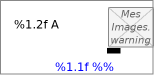
VISUALIZATION VISU_SOURCE_EVAP_COTE_ST10  // 154x75
VAR_IN_OUT
	m_Input_SOURCE : BLOCK_CANON_ST10;
END_VAR
VAR_INPUT
	m_Input_NO_IFIL_RET : Bool;
END_VAR
VAR_INPUT
	m_Input_NO_IEMISS_RET : Bool;
END_VAR
    Polygon (84,73), colour toggle: m_Input_SOURCE.STATE_SRC_ON, invisible if: NOT m_Input_SOURCE.STATE_SRC_ON AND NOT m_Input_SOURCE.STATE_SRC
    Polygon (84,71), invisible if: m_Input_SOURCE.STATE_SRC_ON OR (m_Input_SOURCE.STATE_SRC OR m_Input_SOURCE.STATE_SRC)
    Polygon (70,46)
    Polygon (84,43), invisible if: NOT (m_Input_SOURCE.SRC.STATE_On AND m_Input_SOURCE.HV.STATE_On AND (m_Input_SOURCE.STATE_COURANT>0.0))
    Rectangle (45,60 79x14), "%1.1f %%", text variable: m_Input_SOURCE.STATE_COURANT
    Rectangle (45,36 79x39), invisible if: (NOT m_Input_SOURCE.SRC.AUTOR_ON_IHM AND NOT m_Input_SOURCE.SRC.AUTOR_OFF_IHM) OR NOT PRG_User.ACTU_USER.MAINTENANCE, input disabled if: (NOT m_Input_SOURCE.SRC.AUTOR_ON_IHM AND NOT m_Input_SOURCE.SRC.AUTOR_OFF_IHM) OR NOT PRG_User.ACTU_USER.MAINTENANCE
        OnMouseUp: execute { m_Input_SOURCE.SRC.M_On:=(TRUE); }
    Rectangle (107,48 13x5), colour toggle: m_Input_SOURCE.WATER
    Rectangle (3,18 59x13), "%1.2f A", text variable: m_Input_SOURCE.STATE_I_Fil, invisible if: m_Input_NO_IFIL_RET
    Image (108,7 46x40), invisible if: NOT m_Input_SOURCE.STATE_NOK, image: MesImages.warning
END_VISUALIZATION

(* stored: Version 1.1.0.1, ProductVersion 3.1.4026.18
   Visu VISU_SOURCE_EVAP_COTE_ST10: Id {2e3b1af5-9fe3-481f-a6e6-5545a376b762} *)
